PROGRAM test_prg
VAR
	fb_Blink: FB_Blink;
	triggerBlink : BOOL;
	test_signal : BOOL;
	blinkTime : TIME := T#500MS;
END_VAR

fb_Blink(OnOffTime:= blinkTime, TriggerBlink:= triggerBlink, BlinkSignal=> test_signal);

END_PROGRAM

(* stored: Version 1.1.0.1, ProductVersion 3.1.4024.13
   POU test_prg: Id {dccea0a4-b09a-4ed4-8374-48cd9933971e}, SpecialFunc None *)
